FUNCTION_BLOCK fb_CreateTable
VAR_INPUT
	table:STRING(50);
	bExecute:BOOL;
	DBID:UINT;
	
END_VAR
VAR_OUTPUT
	bError:BOOL:=FALSE;
	bReady:BOOL:=FALSE;
END_VAR
VAR
	sCmd:STRING(255);
	nstep:INT:=10;
	SQLcommand: FB_SQLCommandEvt(sNetid:='',tTimeout:=T#5S);
	Connectdb: FB_sqldatabaseevt(SNetID:='', tTimeout:=T#5S);
	connected:BOOL:=FALSE;
END_VAR

IF bExecute THEN
CASE nstep OF
	10:
		IF connectDB.Connect(DBID) THEN
			
			IF connectdb.bError THEN
				bError:=TRUE;
			ELSE
				connected:=TRUE;	
			END_IF
		END_IF
		IF connected and NOT connectDB.bBusy THEN 
			IF connectDB.CreateCmd(pSQLCommand:= ADR(SQLcommand)) THEN
				nstep:=20;
			END_IF
		END_IF
	20:	
	
		sCmd:=concat('CREATE TABLE ', table);
		sCmd:=concat(sCmd,'(Dátum DATETIME ,
  						temp_set INTEGER ,
  						temp_act INTEGER ,
  						hum_set INTEGER ,
 						 hum_act INTEGER );');
		nstep:=30;
		
	30:
		IF SQLcommand.Execute(pSQLCmd:=ADR(sCmd),
							cbSQLCmd:=SIZEOF(sCmd))
		THEN
			IF sqlcommand.bError THEN
				berror:=TRUE;
			ELSE
			IF NOT SQLcommand.bBusy THEN
				nstep:=40;
			
			END_IF
			END_IF
		END_IF
	40:	
		IF connectDB.Disconnect() THEN
			IF connectdb.bError THEN
				bError:=TRUE;
			ELSE
				connected:=FALSE;
			bReady:=TRUE;
			bExecute:=FALSE;	
		END_IF
		END_IF	
			
END_CASE
END_IF

METHOD Reset : BOOL
VAR_INPUT
END_VAR
bReady:=FALSE;
nstep:=10;
END_METHOD

END_FUNCTION_BLOCK

(* stored: Version 1.1.0.1, ProductVersion 3.1.4024.2
   POU fb_CreateTable: Id {80bf3b00-4ee6-4098-b993-a850821607aa}, SpecialFunc None
   Method Reset: Id {1378e30f-d2df-457e-abcc-716510c6fa4f} *)
